FUNCTION_BLOCK VisionMSGParse (* Tamplate for a simple Basic Function Block Type *)
  (* Standard: 61499-2 *)
  (* Version 0.0, 2018-07-25, 4DIAC-IDE, 4DIAC-Consortium *)
  (* Version 1.0, 2016-05-26, AZ, fortiss GmbH *)
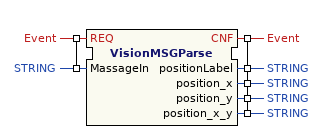
  EVENT_INPUT
    REQ WITH MassageIn; (* Normal Execution Request *)
  END_EVENT
  EVENT_OUTPUT
    CNF WITH positionLabel, position_x, position_y, position_x_y; (* Execution Confirmation *)
  END_EVENT
  VAR_INPUT
    MassageIn : STRING; (* Head+vechlie_x_y+End *)
  END_VAR
  VAR_OUTPUT
    positionLabel : STRING; (* Output event qualifier *)
    position_x : STRING;
    position_y : STRING;
    position_x_y : STRING;
  END_VAR
  VAR
    lastPositionLabel : STRING; (* Internal Variable *)
  END_VAR
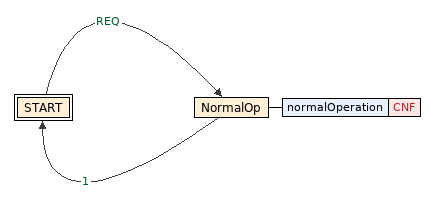
  EC_STATES
    START; (* Initial State *)
    NormalOp : normalOperation -> CNF; (* Normal execution *)
  END_STATES
  EC_TRANSITIONS
    START TO NormalOp := REQ;
    NormalOp TO START := 1;
  END_TRANSITIONS
  ALGORITHM normalOperation IN ST: (* new algorithm *)

  END_ALGORITHM
END_FUNCTION_BLOCK
